Staubli VAL3: find.pgx

public program find(string& x_sItem[] (dimensions=1), bool& x_bFound[] (dimensions=1))
begin
  // check if the item has been foundf
  if save:nBoxType==1
    x_bFound=isDefined(sml:box[x_sItem])
  elseIf save:nBoxType==2
    x_bFound=isDefined(big:box[x_sItem])
  endIf
end
